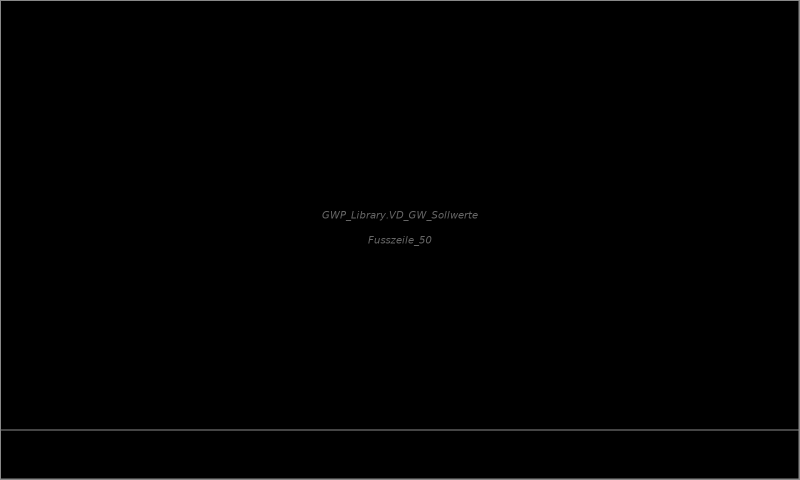
VISUALIZATION VD_GW_Sollwerte  // 800x480
    Frame (0,0 800x430)
        shows GWP_Library.VD_GW_Sollwerte(FB_VD := Main.VD_0)
    Frame (0,0 800x480)
        shows Fusszeile_50()
END_VISUALIZATION

(* stored: Version 1.1.0.1, ProductVersion 3.1.4022.6
   Visu VD_GW_Sollwerte: Id {25133d8d-5b6d-4834-9baf-40b524bfc206} *)
